                   CASE #tempRcvMsgTypeCase OF
                     #MQTT_MSG_TYPE_CONNACK:  // Statement section case 1
                       REGION RECEIVED_CONACK_PACKET    
                         #tempTrcvBufferPos += 1;
                         IF #statRcvBuffer[#tempTrcvBufferPos] = #REMAINING_LEN_2 //remainng Length must be 2;
                         THEN //
                           #tempTrcvBufferPos += 1;
                           //byte one is 0000 000X where X is if Session was set // so depending on clean session or not  evaluate answer of server
                           IF #statRcvBuffer[#tempTrcvBufferPos] = #MQTT_NO_SESSION_PRESENT THEN
                             #tempTrcvBufferPos += 1;
                             //VALID Answer, check code
                             IF #statRcvBuffer[#tempTrcvBufferPos] = #MQTT_CONNACK_ACCEPTED
                             THEN
                               //All good
                               #tempTrcvBufferPos += 1;
                               #tempMqttConnAckRcvStatus := #RESPONSE_GOOD; //evaluate in MQTT StateMachine Below the response
                             ELSE
                               //NOT VALID CONNACK from server shows session has a bad return code
                               #statStatus := #ERR_MQTT_CONNACK_RETURN_CODE_INVALID; // Set correct status that identifies error clearly
                               #statSubfunctionStatus := #statRcvBuffer[#tempTrcvBufferPos]; // Status or return value of called FBs, FCs and system blocks
                               #statFBErrorState := #statFBState; // Set error state number for diagnostic 
                               #statErrorUserCleared := TRUE;
                               // Exit loop
                               EXIT;
                             END_IF;
                           ELSE
                             //NOT VALID, CONNACK from server shows session present
                             #statStatus := #ERR_MQTT_CONNACK_INVALID_SESSION_FLAG; // Set correct status that identifies error clearly
                             #statSubfunctionStatus := #ERR_MQTT_CONNACK_INVALID_SESSION_FLAG; // Status or return value of called FBs, FCs and system blocks
                             #statFBErrorState := #statFBState; // Set error state number for diagnostic 
                             #statErrorUserCleared := TRUE;
                             // Exit loop
                             EXIT;
                           END_IF;
                         ELSE // We got a CONNACK paket, but remaining length was not 2 (Error)
                           #statStatus := #ERR_MQTT_REM_LEN_INVALID; // Set correct status that identifies error clearly
                           #statSubfunctionStatus := #ERR_MQTT_REM_LEN_INVALID; // Status or return value of called FBs, FCs and system blocks
                           #statFBErrorState := #statFBState; // Set error state number for diagnostic 
                           #statErrorUserCleared := TRUE;
                           // Exit loop
                           EXIT;
                         END_IF;
                       END_REGION RECEIVED_CONACK_PACKET  
                     #MQTT_MSG_TYPE_PINGRESP:
                       REGION RECEIVED_PINGRESP_PAKET
                         #tempTrcvBufferPos += 1;
                         IF #statRcvBuffer[#tempTrcvBufferPos] = #REMAINIG_LEN_0 //remainng Length must be 0;
                         THEN
                           #tempTrcvBufferPos += 1;
                           #tempMqttPingRspRcv := #RESPONSE_GOOD; //evaluate in MQTT StateMachine Below the response
                         ELSE// We got a Pingrsp paket, but remaining length was not 0 (Error)
                           #statStatus := #ERR_MQTT_REM_LEN_INVALID; // Set correct status that identifies error clearly
                           #statSubfunctionStatus := #ERR_MQTT_REM_LEN_INVALID; // Status or return value of called FBs, FCs and system blocks
                           #statFBErrorState := #statFBState; // Set error state number for diagnostic 
                           #statErrorUserCleared := TRUE;
                           // Exit loop
                           EXIT;
                         END_IF;
                       END_REGION RECEIVED_PINGRESP_PAKET
                     #MQTT_MSG_TYPE_PUBACK:
                       REGION RECEIVED_PUBACK_PAKET
                         #tempTrcvBufferPos += 1;
                         IF #statRcvBuffer[#tempTrcvBufferPos] = #REMAINING_LEN_2 //remainng Length must be 2;
                         THEN //
                           #tempTrcvBufferPos += 1;
                           #tempWordForSliceAddress := UINT_TO_WORD(#statPaketId);
                           IF #statRcvBuffer[#tempTrcvBufferPos] = #tempWordForSliceAddress.%B1 THEN
                             #tempTrcvBufferPos += 1;
                             IF #statRcvBuffer[#tempTrcvBufferPos] = #tempWordForSliceAddress.%B0 THEN
                               #tempTrcvBufferPos += 1;
                               #tempMqttPubAckRcv := #RESPONSE_GOOD;
                             ELSE
                               #tempTrcvBufferPos += 1;
                               #tempMqttPubAckRcv := #RESPONSE_PAKET_ID_INVALID;
                             END_IF;
                           ELSE
                             #tempTrcvBufferPos += 1;
                             #tempMqttPubAckRcv := #RESPONSE_PAKET_ID_INVALID;
                           END_IF;
                         ELSE
                           #statStatus := #ERR_MQTT_REM_LEN_INVALID; // Set correct status that identifies error clearly
                           #statSubfunctionStatus := #ERR_MQTT_REM_LEN_INVALID; // Status or return value of called FBs, FCs and system blocks
                           #statFBErrorState := #statFBState; // Set error state number for diagnostic 
                           #statErrorUserCleared := TRUE;
                           // Exit loop
                           EXIT;
                         END_IF;
                       END_REGION RECEIVED_PUBACK_PAKET
                     #MQTT_MSG_TYPE_PUBREC:
                       REGION RECEIVED_PUBREC_PAKET
                         #tempTrcvBufferPos += 1;
                         IF #statRcvBuffer[#tempTrcvBufferPos] = #REMAINING_LEN_2 //remainng Length must be 2;
                         THEN //
                           #tempTrcvBufferPos += 1;
                           #tempWordForSliceAddress := UINT_TO_WORD(#statPaketId);
                           IF #statRcvBuffer[#tempTrcvBufferPos] = #tempWordForSliceAddress.%B1 THEN
                             #tempTrcvBufferPos += 1;
                             IF #statRcvBuffer[#tempTrcvBufferPos] = #tempWordForSliceAddress.%B0 THEN
                               #tempTrcvBufferPos += 1;
                               #tempMqttPubRecRcv := #RESPONSE_GOOD;
                             ELSE
                               #tempTrcvBufferPos += 1;
                               #tempMqttPubRecRcv := #RESPONSE_PAKET_ID_INVALID;
                             END_IF;
                           ELSE
                             #tempTrcvBufferPos += 1;
                             #tempMqttPubRecRcv := #RESPONSE_PAKET_ID_INVALID;
                           END_IF;
                         ELSE
                           #statStatus := #ERR_MQTT_REM_LEN_INVALID; // Set correct status that identifies error clearly
                           #statSubfunctionStatus := #ERR_MQTT_REM_LEN_INVALID; // Status or return value of called FBs, FCs and system blocks
                           #statFBErrorState := #statFBState; // Set error state number for diagnostic 
                           #statErrorUserCleared := TRUE;
                           // Exit loop
                           EXIT;
                         END_IF;
                       END_REGION RECEIVED_PUBREC_PAKET
                     #MQTT_MSG_TYPE_PUBCOMP:
                       REGION RECEIVED_PUBCOMP_PAKET
                         #tempTrcvBufferPos += 1;
                         IF #statRcvBuffer[#tempTrcvBufferPos] = #REMAINING_LEN_2 //remainng Length must be 2;
                         THEN //
                           #tempTrcvBufferPos += 1;
                           #tempWordForSliceAddress := UINT_TO_WORD(#statPaketId);
                           IF #statRcvBuffer[#tempTrcvBufferPos] = #tempWordForSliceAddress.%B1 THEN
                             #tempTrcvBufferPos += 1;
                             IF #statRcvBuffer[#tempTrcvBufferPos] = #tempWordForSliceAddress.%B0 THEN
                               #tempTrcvBufferPos += 1;
                               #tempMqttPubCompRcv := #RESPONSE_GOOD;
                             ELSE
                               #tempTrcvBufferPos += 1;
                               #tempMqttPubCompRcv := #RESPONSE_PAKET_ID_INVALID;
                             END_IF;
                           ELSE
                             #tempTrcvBufferPos += 1;
                             #tempMqttPubCompRcv := #RESPONSE_PAKET_ID_INVALID;
                           END_IF;
                         ELSE
                           #statStatus := #ERR_MQTT_REM_LEN_INVALID; // Set correct status that identifies error clearly
                           #statSubfunctionStatus := #ERR_MQTT_REM_LEN_INVALID; // Status or return value of called FBs, FCs and system blocks
                           #statFBErrorState := #statFBState; // Set error state number for diagnostic 
                           #statErrorUserCleared := TRUE;
                           // Exit loop
                           EXIT;
                         END_IF;
                       END_REGION RECEIVED_PUBCOMP_PAKET
                     #MQTT_MSG_TYPE_SUBACK:
                       REGION RECEIVED_SUBACK_PAKET
                         #tempTrcvBufferPos += 1;
                         IF #statRcvBuffer[#tempTrcvBufferPos] = #REMAINING_LEN_3 //remainng Length must be 3;
                         THEN //
                           #tempTrcvBufferPos += 1;
                           #tempWordForSliceAddress := UINT_TO_WORD(#statPaketId);
                           IF #statRcvBuffer[#tempTrcvBufferPos] = #tempWordForSliceAddress.%B1 THEN
                             #tempTrcvBufferPos += 1;
                             IF #statRcvBuffer[#tempTrcvBufferPos] = #tempWordForSliceAddress.%B0 THEN
                               #tempTrcvBufferPos += 1;
                               IF #statRcvBuffer[#tempTrcvBufferPos] = #SUBSCRIBE_FAILURE THEN
                                 #tempTrcvBufferPos += 1;
                                 #tempMqttSubAckRcv := #RESPONSE_SUBSCRIBE_FAILED;
                               ELSE
                                 #tempTrcvBufferPos += 1;
                                 #tempMqttSubAckRcv := #RESPONSE_GOOD;
                               END_IF;
                             ELSE
                               #tempTrcvBufferPos += 1;
                               #tempMqttSubAckRcv := #RESPONSE_PAKET_ID_INVALID;
                             END_IF;
                           ELSE
                             #tempTrcvBufferPos += 1;
                             #tempMqttSubAckRcv := #RESPONSE_PAKET_ID_INVALID;
                           END_IF;
                         ELSE
                           #statStatus := #ERR_MQTT_REM_LEN_INVALID; // Set correct status that identifies error clearly
                           #statSubfunctionStatus := #ERR_MQTT_REM_LEN_INVALID; // Status or return value of called FBs, FCs and system blocks
                           #statFBErrorState := #statFBState; // Set error state number for diagnostic 
                           #statErrorUserCleared := TRUE;
                           // Exit loop
                           EXIT;
                         END_IF;
                       END_REGION RECEIVED_SUBACK_PAKET
                     #MQTT_MSG_TYPE_UNSUBACK:
                       REGION RECEIVED_UNSUBACK_PAKET
                         #tempTrcvBufferPos += 1;
                         IF #statRcvBuffer[#tempTrcvBufferPos] = #REMAINING_LEN_2 //remainng Length must be 2;
                         THEN //
                           #tempTrcvBufferPos += 1;
                           #tempWordForSliceAddress := UINT_TO_WORD(#statPaketId);
                           IF #statRcvBuffer[#tempTrcvBufferPos] = #tempWordForSliceAddress.%B1 THEN
                             #tempTrcvBufferPos += 1;
                             IF #statRcvBuffer[#tempTrcvBufferPos] = #tempWordForSliceAddress.%B0 THEN
                               #tempTrcvBufferPos += 1;
                               #tempMqttUnSubAckRcv := #RESPONSE_GOOD;
                             ELSE
                               #tempTrcvBufferPos += 1;
                               #tempMqttUnSubAckRcv := #RESPONSE_PAKET_ID_INVALID;
                             END_IF;
                           ELSE
                             #tempTrcvBufferPos += 1;
                             #tempMqttUnSubAckRcv := #RESPONSE_PAKET_ID_INVALID;
                           END_IF;
                         ELSE
                           #statStatus := #ERR_MQTT_REM_LEN_INVALID; // Set correct status that identifies error clearly
                           #statSubfunctionStatus := #ERR_MQTT_REM_LEN_INVALID; // Status or return value of called FBs, FCs and system blocks
                           #statFBErrorState := #statFBState; // Set error state number for diagnostic 
                           #statErrorUserCleared := TRUE;
                           // Exit loop
                           EXIT;
                         END_IF;
                       END_REGION RECEIVED_UNSUBACK_PAKET
                     #MQTT_MSG_TYPE_RCV_PUB_MESSAGE:
                       REGION RECEIVED_PUBLISH_PAKET_FROM_BROKER
                         //Received a message, start process.
                         //init
                         #tempMultiplierToDecode := #INIT_UDINT_1;
                         #statRcvMsgInternalStatus := #MSG_DECODE_STATUS_NO_NEW_MSG;
                         #statRcvMsgTotalLen := 0;
                         #statRcvMsgTopicLen := 0;
                         #statRcvMsgPayloadLen := 0;
                         //Check and store QoS for later use
                         IF (#statRcvBuffer[#tempTrcvBufferPos] AND #BIT_MASK_QOS) = #MQTT_MSG_TYPE_RCV_PUB_MESSAGE_QoS0
                         THEN
                           #statRcvMsgQoS := #MQTT_QOS_0;
                         ELSIF (#statRcvBuffer[#tempTrcvBufferPos] AND #BIT_MASK_QOS) = #MQTT_MSG_TYPE_RCV_PUB_MESSAGE_QoS1
                         THEN
                           #statRcvMsgQoS := #MQTT_QOS_1;
                         ELSIF (#statRcvBuffer[#tempTrcvBufferPos] AND #BIT_MASK_QOS) = #MQTT_MSG_TYPE_RCV_PUB_MESSAGE_QoS2
                         THEN
                           #statRcvMsgQoS := #MQTT_QOS_2;
                         ELSIF (#statRcvBuffer[#tempTrcvBufferPos] AND #BIT_MASK_QOS) = #MQTT_MSG_TYPE_RCV_PUB_MESSAGE_BAD
                         THEN
                           #statStatus := #ERR_MQTT_MALFORMED_QOS_RECEIVED; // Set correct status that identifies error clearly
                           #statSubfunctionStatus := #ERR_MQTT_MALFORMED_QOS_RECEIVED; // Status or return value of called FBs, FCs and system blocks
                           #statFBErrorState := #statFBState; // Set error state number for diagnostic 
                           #statErrorUserCleared := TRUE;
                           // Exit loop
                           EXIT;
                         END_IF;

                         //Calculate total publish len (topic,paketid,payload)
                         REPEAT
                           #tempTrcvBufferPos += 1; //Increment
                           #statRcvMsgTotalLen += BYTE_TO_UDINT((#statRcvBuffer[#tempTrcvBufferPos] AND #DEFAULT_MULTIPLIER_BYTE_127)) * #tempMultiplierToDecode;
                           #tempMultiplierToDecode *= #SEND_LEN_MULTIPLIER_UDINT_128;
                           IF (#tempMultiplierToDecode > #MAX_ALLOWED_PAKET_SIZE)
                           THEN//Throw error here // Malformed remain length.
                             #statStatus := #ERR_MQTT_REM_LEN_INVALID; // Set correct status that identifies error clearly
                             #statSubfunctionStatus := #ERR_MQTT_REM_LEN_INVALID; // Status or return value of called FBs, FCs and system blocks
                             #statFBErrorState := #statFBState; // Set error state number for diagnostic 
                             #statErrorUserCleared := TRUE;
                             // Exit loop
                             EXIT;
                           END_IF;
                         UNTIL ((#statRcvBuffer[#tempTrcvBufferPos] AND UDINT_TO_BYTE(#SEND_LEN_MULTIPLIER_UDINT_128)) = 0)
                         END_REPEAT;
                         #tempTrcvBufferPos += 1; //Increment
                         //#statIncPaketRemLen contains total paket len
                         //Save Topic Len
                         #tempWordForSliceAddress.%B1 := #statRcvBuffer[#tempTrcvBufferPos]; //MSB
                         #tempTrcvBufferPos += 1; //Increment
                         #tempWordForSliceAddress.%B0 := #statRcvBuffer[#tempTrcvBufferPos]; //LSB
                         #tempTrcvBufferPos += 1; //Increment
                         #statRcvMsgTopicLen := WORD_TO_UINT(#tempWordForSliceAddress);
                         //Set Payload len
                         IF #statRcvMsgQoS = #MQTT_QOS_0 THEN
                           //Payload Len is total Len minus topic len minus topic len info 
                           #statRcvMsgPayloadLen := #statRcvMsgTotalLen - #statRcvMsgTopicLen - #TWO_BYTE_LEN_INFO;
                         ELSE
                           //PayloadLen is total Len minus topic len minus topic len info minus paket Id len
                           #statRcvMsgPayloadLen := #statRcvMsgTotalLen - #statRcvMsgTopicLen - #TWO_BYTE_LEN_INFO - #TWO_BYTE_LEN_INFO;
                         END_IF;

                         //Clear Output message:
                         #receivedTopic := #EMPTY_WSTRING;
                         //Start receiving with topic
                         #statRcvMsgDecodeState := #MSG_DECODE_STATE_TOPIC;
                         //Start Topic at first character
                         #statRcvMsgTopicPos := #FIRST_CHARACTER;
                         //Start RcvMsg at first array element
                         #statRcvMsgPayloadPos := LOWER_BOUND(ARR := #receivedMsgPayload, DIM := #ONE_DIMENSION);
                         //Set Output for received len according to array dimension
                         #tempReceivedMsgDataArrayTotalLen := ABS(UPPER_BOUND(ARR := #receivedMsgPayload, DIM := #ONE_DIMENSION) - LOWER_BOUND(ARR := #receivedMsgPayload, DIM := #ONE_DIMENSION)) + #ARRAY_LEN_OFFSET_PLUS_1;
                         IF #statRcvMsgPayloadLen < #tempReceivedMsgDataArrayTotalLen THEN
                           #statRcvMsgDataLen := #statRcvMsgPayloadLen;
                         ELSE
                           #statRcvMsgDataLen := DINT_TO_UDINT(#tempReceivedMsgDataArrayTotalLen);
                         END_IF;
                       END_REGION RECEIVED_PUBLISH_PAKET_FROM_BROKER
                     #MQTT_MSG_DECODING:
                       REGION RECEIVED_PAKET_DECODE
                         CASE #statRcvMsgDecodeState OF
                           #MSG_DECODE_STATE_NO_PROCESSING: // NO Processing
                             ;
                           #MSG_DECODE_STATE_TOPIC:  // Statement section case 1
                             #tempReceivedTopicStringMaxLen := MAX_LEN(#receivedTopic);
                             //Copy Topic To WString Inout
                             IF #statRcvMsgTopicPos <= #tempReceivedTopicStringMaxLen THEN
                               #receivedTopic[#statRcvMsgTopicPos] := BYTE_TO_WCHAR(#statRcvBuffer[#tempTrcvBufferPos]);
                               #statRcvMsgTopicPos += 1;
                             ELSE
                               //Max String len reached.
                               #statRcvMsgInternalStatus := #MSG_DECODE_STATUS_TOPIC_TOO_LONG;
                             END_IF;
                             //decrement
                             #statRcvMsgTopicLen -= 1;
                             //increment
                             #tempTrcvBufferPos += 1;
                             //Check condition, if topic fully decoded:
                             IF #statRcvMsgTopicLen <= 0 THEN
                               //Decide what to do next:
                               IF #statRcvMsgQoS > #MQTT_QOS_0 THEN
                                 //NextStep Decode PaketID
                                 #statRcvMsgDecodeState := #MSG_DECODE_STATE_PAKET_ID_MSB;
                               ELSIF #statRcvMsgQoS = #MQTT_QOS_0 AND #statRcvMsgPayloadLen > 0 THEN
                                 //NextStep Decode Payload
                                 #statRcvMsgDecodeState := #MSG_DECODE_STATE_PAYLOAD;
                               ELSE
                                 // QoS=0 and no Payload => Done
                                 // Decoding complete
                                 #statRcvMsgDecodeState := #MSG_DECODE_STATE_NO_PROCESSING;
                                 //Set New message flag
                                 IF #statRcvMsgInternalStatus = #MSG_DECODE_STATUS_NO_NEW_MSG THEN
                                   //New message received ok
                                   #statRcvMsgStatus := #MSG_DECODE_STATUS_NEW_MSG_OK;
                                 ELSE
                                   //Message received, but Payload or Topic longer than inout data area
                                   #statRcvMsgStatus := #MSG_DECODE_STATUS_TOPIC_TOO_LONG;
                                 END_IF;
                               END_IF;
                             END_IF;
                           #MSG_DECODE_STATE_PAKET_ID_MSB:  // Decode PaketId MSB
                             //Copy PaketID
                             #statRcvMsgPaketId.%B1 := #statRcvBuffer[#tempTrcvBufferPos]; //MSB
                             #tempTrcvBufferPos += 1; //Increment
                             #statRcvMsgDecodeState := #MSG_DECODE_STATE_PAKET_ID_LSB;
                           #MSG_DECODE_STATE_PAKET_ID_LSB: // Decode PaketId LSB
                             //Copy PaketID
                             #statRcvMsgPaketId.%B0 := #statRcvBuffer[#tempTrcvBufferPos]; //LSB
                             #tempTrcvBufferPos += 1; //Increment
                             IF #statRcvMsgPayloadLen > 0 THEN
                               #statRcvMsgDecodeState := #MSG_DECODE_STATE_PAYLOAD;
                             ELSE
                               // Decoding complete
                               #statRcvMsgDecodeState := #MSG_DECODE_STATE_NO_PROCESSING;
                               //Set New message flag
                               IF #statRcvMsgInternalStatus = #MSG_DECODE_STATUS_NO_NEW_MSG THEN
                                 //New message received ok
                                 #statRcvMsgStatus := #MSG_DECODE_STATUS_NEW_MSG_OK;
                               ELSE
                                 //Message received, but Payload or Topic longer than inout data area
                                 #statRcvMsgStatus := #MSG_DECODE_STATUS_TOPIC_TOO_LONG;
                               END_IF;
                               // Send PubAck Msg
                               #statSendPubAckMsg := TRUE;
                             END_IF;
                           #MSG_DECODE_STATE_PAYLOAD:
                             #tempUpperBoundRcvMsgDataArray := UPPER_BOUND(ARR := #receivedMsgPayload, DIM := #ONE_DIMENSION);

                             IF #statRcvMsgPayloadPos <= #tempUpperBoundRcvMsgDataArray THEN
                               //Copy to output
                               #receivedMsgPayload[#statRcvMsgPayloadPos] := (#statRcvBuffer[#tempTrcvBufferPos]);
                               //Increment the pos
                               #statRcvMsgPayloadPos += 1;
                             ELSE
                               //Max Payload len reached, skip
                               #statRcvMsgInternalStatus := #MSG_DECODE_STATUS_PAYLOAD_TOO_LONG;
                             END_IF;
                             //Decrement msg payload len
                             #statRcvMsgPayloadLen -= 1;
                             //Increment Buffer Pos
                             #tempTrcvBufferPos += 1;
                             //Check condition, if payload fully decoded:
                             IF #statRcvMsgPayloadLen <= 0 THEN
                               // Decoding complete
                               #statRcvMsgDecodeState := #MSG_DECODE_STATE_NO_PROCESSING;
                               //Set New message flag
                               IF #statRcvMsgInternalStatus = #MSG_DECODE_STATUS_NO_NEW_MSG THEN
                                 //New message received ok
                                 #statRcvMsgStatus := #MSG_DECODE_STATUS_NEW_MSG_OK;
                               ELSE
                                 //Message received, but Payload or Topic longer than inout data area
                                 #statRcvMsgStatus := #MSG_DECODE_STATUS_PAYLOAD_TOO_LONG;
                               END_IF;
                               //Decide if a PUB ACK needs to be send
                               IF #statRcvMsgQoS > #MQTT_QOS_0 THEN
                                 // Send PubAck Msg
                                 #statSendPubAckMsg := TRUE;
                               END_IF;
                             END_IF;
                           ELSE
                             //else case
                             #statStatus := #ERR_UNDEFINED_STATE;
                             #statErrorUserCleared := TRUE;
                             ;
                         END_CASE;
                       END_REGION RECEIVED_PAKET_DECODE
                     ELSE // No Header found, SKIP entry of buffer:
                       #tempTrcvBufferPos += 1;
                   END_CASE;
                 END_WHILE;
               END_REGION TRCV_NEW_DATA
             END_IF;

             //Send an Publish Acknowledge Msg, if necessary
             REGION SEND_PUB_ACK_MSG_ON_SUBSCRIPTIONS
               //Send Acknowledgements to Subscribed messages, if requested (QoS =1)
               IF #statSendPubAckMsg = TRUE AND // send pub ack Request
                 #statMqttCommandState = #MQTT_COMMAND_STATE_NO_PROCESSING AND // no send job processing
                 #tempTsendcBusy = FALSE AND // tsendC is ready
                 #tempTsendcDone = FALSE // tsendC did not finished in this cycle
               THEN
                 //Set Pos
                 #statSendBufferPos := 0;
                 //Write Msg Type
                 #statSendBuffer[#statSendBufferPos] := #MQTT_MSG_TYPE_PUBACK;
                 #statSendBufferPos += 1;
                 //Write Msg Len
                 #statSendBuffer[#statSendBufferPos] := #REMAINING_LEN_2;
                 #statSendBufferPos += 1;
                 //Write Paket Id - first MSB then LSB
                 #statSendBuffer[#statSendBufferPos] := #statRcvMsgPaketId.%B1;
                 #statSendBufferPos += 1;
                 #statSendBuffer[#statSendBufferPos] := #statRcvMsgPaketId.%B0;
                 #statSendBufferPos += 1;
                 //Set Send Len:
                 #statTsendcLen := #statSendBufferPos;
                 //Send msg
                 #statTsendcReq := TRUE;
                 //Reset ack:
                 #statSendPubAckMsg := FALSE;
               END_IF;
             END_REGION SEND_PUB_ACK_MSG_ON_SUBSCRIPTIONS

             REGION MQTT_STATE_MACHINE
               CASE #statMqttConnectState OF
                 #MQTT_CONNECT_STATE_NO_PROCESSING:  // Statement section case 1
                   ;
                 #MQTT_CONNECT_STATE_BUILD_PAKET:  //
                   REGION BUILD_CONNECT_PAKET
                     //Remaining Length is the length of the variable header (10 bytes) plus the length of the Payload. 
                     //Max Len of Mqtt pakets is per Standard 268,435,455 Bytes (ff,ff,ff,7f)
                     //Calculate Remain Len will be 10 bytes
                     //plus Len of ClientId   (max 3*16382 WChars= 49.146 Bytes)
                     //plus Len of User (max 3*16382 WChars= 49.146 Bytes)
                     //plus Len of PW (max 3*16382 WChars= 49.146 Bytes)
                     //plus Len of WillTopic (max 3*16382 WChars= 49.146 Bytes)
                     //plus Len of WillMessage (max 65535 Bytes - as only 2 Bytes Len info is possible)
                     // = Total 262 119 Bytes


                     // Must obey, if not currently sending PubAck Msg on a subscription
                     // Else, try in the next cycle
                     IF #tempTsendcBusy = FALSE AND // tsendC is ready
                       #tempTsendcDone = FALSE AND  // tsendC did not finish in this cycle
                       #statTsendcReq = FALSE THEN // no request from pub ack request

                       //Only need to encode header once
                       IF #statPaketHeaderEncodeDone = FALSE THEN
                         // INIT
                         #statSendBufferPos := 0;
                         #statClientIdPos := #FIRST_CHARACTER;
                         #statClientIdEncodeState := #FIRST_ENCODING;

                         #statWillTopicEncodeState := #FIRST_ENCODING;
                         #statWillTopicPos := #FIRST_CHARACTER;

                         #statWillMessageEncodeState := #FIRST_ENCODING;
                         #statWillMessagePos := 0; // The Posistion for the WILL Message Array

                         #statUserNameEncodeState := #FIRST_ENCODING;
                         #statUserNamePos := #FIRST_CHARACTER;

                         #statPasswordEncodeState := #FIRST_ENCODING;
                         #statPasswordPos := #FIRST_CHARACTER;

                         #statSendPaketTotalRemLen := #CONNECT_HEADER_10BYTE_LEN;
                         #statClientIdLenUtf8Encoded := 0;
                         #statWillTopicLenUtf8Encoded := 0;
                         #statUsernameLenUtf8Encoded := 0;
                         #statPasswordLenUtf8Encoded := 0;
                         //End Init

                         // Encode Client ID Len
                         // Client ID must always be present
                         FOR #tempLoopCounter := #FIRST_CHARACTER TO LEN(#clientIdentifier) DO
                           "LMQTT_ConvertToUtf8"(character     := #clientIdentifier[#tempLoopCounter],
                                                 convertedUtf8 => #tempConvertedUtf8,
                                                 bytesUsed     => #tempBytesUsedUtf8,
                                                 error         => #tempErrorConvertUtf8,
                                                 status        => #tempStatusConvertUtf8);
                           #statClientIdLenUtf8Encoded := #statClientIdLenUtf8Encoded + #tempBytesUsedUtf8;
                         END_FOR;

                         #statSendPaketTotalRemLen := #statSendPaketTotalRemLen + #statClientIdLenUtf8Encoded + #TWO_BYTE_LEN_INFO;


                         IF #username <> #EMPTY_WSTRING
                         THEN
                           #tempUserFlag := TRUE;
                           FOR #tempLoopCounter := #FIRST_CHARACTER TO LEN(#username) DO
                             "LMQTT_ConvertToUtf8"(character     := #username[#tempLoopCounter],
                                                   convertedUtf8 => #tempConvertedUtf8,
                                                   bytesUsed     => #tempBytesUsedUtf8,
                                                   error         => #tempErrorConvertUtf8,
                                                   status        => #tempStatusConvertUtf8);
                             #statUsernameLenUtf8Encoded := #statUsernameLenUtf8Encoded + #tempBytesUsedUtf8;
                           END_FOR;
                           #statSendPaketTotalRemLen := #statSendPaketTotalRemLen + #statUsernameLenUtf8Encoded + #TWO_BYTE_LEN_INFO;
                         ELSE
                           #statUserNameEncodeState := #NOT_USED_NO_ENCODING;
                           #tempUserFlag := FALSE;
                         END_IF;

                         IF #password <> #EMPTY_WSTRING AND #username <> #EMPTY_WSTRING
                         THEN
                           #tempPasswordFlag := TRUE;
                           FOR #tempLoopCounter := #FIRST_CHARACTER TO LEN(#password) DO
                             "LMQTT_ConvertToUtf8"(character     := #password[#tempLoopCounter],
                                                   convertedUtf8 => #tempConvertedUtf8,
                                                   bytesUsed     => #tempBytesUsedUtf8,
                                                   error         => #tempErrorConvertUtf8,
                                                   status        => #tempStatusConvertUtf8);
                             #statPasswordLenUtf8Encoded := #statPasswordLenUtf8Encoded + #tempBytesUsedUtf8;
                           END_FOR;
                           #statSendPaketTotalRemLen := #statSendPaketTotalRemLen + #statPasswordLenUtf8Encoded + #TWO_BYTE_LEN_INFO;
                         ELSE
                           #statPasswordEncodeState := #NOT_USED_NO_ENCODING;
                           #tempPasswordFlag := FALSE;
                         END_IF;


                         IF #willtopic <> #EMPTY_WSTRING
                         THEN
                           #tempWillFlag := TRUE;
                           CASE #statWillQos OF
                             #MQTT_QOS_0:  // Statement section case 1
                               #tempWillQoS1 := FALSE;
                               #tempWillQoS2 := FALSE;
                             #MQTT_QOS_1:  // Statement section case 2 to 4
                               #tempWillQoS1 := TRUE;
                               #tempWillQoS2 := FALSE;
                             #MQTT_QOS_2:
                               #tempWillQoS1 := FALSE;
                               #tempWillQoS2 := True;
                             ELSE  // Statement section ELSE
                               ;
                           END_CASE;
                           FOR #tempLoopCounter := #FIRST_CHARACTER TO LEN(#willtopic) DO
                             // Statement section FOR
                             "LMQTT_ConvertToUtf8"(character     := #willtopic[#tempLoopCounter],
                                                   convertedUtf8 => #tempConvertedUtf8,
                                                   bytesUsed     => #tempBytesUsedUtf8,
                                                   error         => #tempErrorConvertUtf8,
                                                   status        => #tempStatusConvertUtf8);
                             #statWillTopicLenUtf8Encoded := #statWillTopicLenUtf8Encoded + #tempBytesUsedUtf8;
                           END_FOR;
                           //Add WillTopic Len and Will Message Len (and len info twice)
                           #statSendPaketTotalRemLen := #statSendPaketTotalRemLen + #statWillTopicLenUtf8Encoded + #statWillMessageCnt + (2 * #TWO_BYTE_LEN_INFO);
                         ELSE
                           #statWillTopicEncodeState := #NOT_USED_NO_ENCODING;
                           #statWillMessageEncodeState := #NOT_USED_NO_ENCODING;
                           #tempWillFlag := FALSE;
                           #statWillRetain := FALSE;
                           #tempWillQoS1 := FALSE;
                           #tempWillQoS2 := FALSE;
                         END_IF;

                         //Build Connect Telegram
                         //Fixed Header - Write Paket Type
                         #statSendBuffer[#statSendBufferPos] := #MQTT_MSG_TYPE_CONNECT; // 1 Byte
                         #statSendBufferPos += 1; // increment

                         //Write Remaining Paket Len info 
                         WHILE (#statSendPaketTotalRemLen > #DEFAULT_VALUE_ZERO)
                         DO//See MQTT Spec for explanation of this calculation
                           #statEncodedRemPaketLenAsByte := UDINT_TO_BYTE(#statSendPaketTotalRemLen MOD #SEND_LEN_MULTIPLIER_UDINT_128);
                           #statSendPaketTotalRemLen := #statSendPaketTotalRemLen / #SEND_LEN_MULTIPLIER_UDINT_128;
                           // if there are more data to encode, set the top bit of this byte
                           IF #statSendPaketTotalRemLen > #DEFAULT_VALUE_ZERO
                           THEN
                             // Do this and continue while loop
                             #statEncodedRemPaketLenAsByte := #statEncodedRemPaketLenAsByte OR UDINT_TO_BYTE(#SEND_LEN_MULTIPLIER_UDINT_128);
                             #statSendBuffer[#statSendBufferPos] := #statEncodedRemPaketLenAsByte;
                             #statSendBufferPos += 1;
                           ELSE
                             //do this and leave while loop
                             #statSendBuffer[#statSendBufferPos] := #statEncodedRemPaketLenAsByte;
                             #statSendBufferPos += 1;
                           END_IF;
                         END_WHILE;

                         //Build Connect Telegram
                         // Write Protocol name
                         #statSendBuffer[#statSendBufferPos] := #CONN_PROTOCOL_NAME_0;
                         #statSendBufferPos += 1;
                         #statSendBuffer[#statSendBufferPos] := #CONN_PROTOCOL_NAME_4;
                         #statSendBufferPos += 1;
                         #statSendBuffer[#statSendBufferPos] := CHAR_TO_BYTE('M');
                         #statSendBufferPos += 1;
                         #statSendBuffer[#statSendBufferPos] := CHAR_TO_BYTE('Q');
                         #statSendBufferPos += 1;
                         #statSendBuffer[#statSendBufferPos] := CHAR_TO_BYTE('T');
                         #statSendBufferPos += 1;
                         #statSendBuffer[#statSendBufferPos] := CHAR_TO_BYTE('T');
                         #statSendBufferPos += 1;
                         //Write Protocol Level
                         #statSendBuffer[#statSendBufferPos] := #CONN_PROTOCOL_MQTT_VERSION_3_1_1;
                         #statSendBufferPos += 1;
                         //Write Connect Flags
                         #statSendBuffer[#statSendBufferPos].%X0 := false;
                         #statSendBuffer[#statSendBufferPos].%X1 := True;
                         #statSendBuffer[#statSendBufferPos].%X2 := #tempWillFlag;
                         #statSendBuffer[#statSendBufferPos].%X3 := #tempWillQoS1;
                         #statSendBuffer[#statSendBufferPos].%X4 := #tempWillQoS2;
                         #statSendBuffer[#statSendBufferPos].%X5 := #statWillRetain;
                         #statSendBuffer[#statSendBufferPos].%X6 := #tempPasswordFlag;
                         #statSendBuffer[#statSendBufferPos].%X7 := #tempUserFlag;
                         #statSendBufferPos += 1;
                         //Write Keep Alive in sec
                         #tempWordForSliceAddress := UINT_TO_WORD(#connParam.keepAlive);
                         #statSendBuffer[#statSendBufferPos] := #tempWordForSliceAddress.%B1;
                         #statSendBufferPos += 1;
                         #statSendBuffer[#statSendBufferPos] := #tempWordForSliceAddress.%B0;
                         #statSendBufferPos += 1;

                         //Set To Complete this, can skip in further progess
                         #statPaketHeaderEncodeDone := TRUE;
                       END_IF;

                       // Payload
                       // These fields, if present, MUST appear in the order:
                       // Client Identifier, Will topic, Will message, User Name, password


                       //ClientIdentifier
                       IF #statSendBufferPos <= #MAX_BUFFER_LEN_SEND - #TWO_BYTE_LEN_INFO THEN
                         CASE #statClientIdEncodeState OF
                           #FIRST_ENCODING:  // Statement section case 1
                             //ADD len info into paket

                             #tempWordForSliceAddress := UINT_TO_WORD(#statClientIdLenUtf8Encoded);
                             #statSendBuffer[#statSendBufferPos] := #tempWordForSliceAddress.%B1; //MSB
                             #statSendBufferPos += 1;
                             #statSendBuffer[#statSendBufferPos] := #tempWordForSliceAddress.%B0; // LSB
                             #statSendBufferPos += 1;

                             FOR #tempLoopCounter := #statClientIdPos TO LEN(#clientIdentifier) DO
                               "LMQTT_ConvertToUtf8"(character     := #clientIdentifier[#tempLoopCounter],
                                                     convertedUtf8 => #tempConvertedUtf8,
                                                     bytesUsed     => #tempBytesUsedUtf8,
                                                     error         => #tempErrorConvertUtf8,
                                                     status        => #tempStatusConvertUtf8);

                               IF #statSendBufferPos + #tempBytesUsedUtf8 <= #MAX_BUFFER_LEN_SEND THEN
                                 #statClientIdPos += 1;
                                 CASE #tempBytesUsedUtf8 OF
                                   #UTF_1_BYTE_USED:  // Statement section case 1
                                     #statSendBuffer[#statSendBufferPos] := #tempConvertedUtf8.%B0;
                                     #statSendBufferPos += 1;
                                   #UTF_2_BYTE_USED:
                                     #statSendBuffer[#statSendBufferPos] := #tempConvertedUtf8.%B0;
                                     #statSendBufferPos += 1;
                                     #statSendBuffer[#statSendBufferPos] := #tempConvertedUtf8.%B1;
                                     #statSendBufferPos += 1;
                                   #UTF_3_BYTE_USED:  // Statement section case 2 to 4
                                     #statSendBuffer[#statSendBufferPos] := #tempConvertedUtf8.%B0;
                                     #statSendBufferPos += 1;
                                     #statSendBuffer[#statSendBufferPos] := #tempConvertedUtf8.%B1;
                                     #statSendBufferPos += 1;
                                     #statSendBuffer[#statSendBufferPos] := #tempConvertedUtf8.%B2;
                                     #statSendBufferPos += 1;
                                   ELSE  // Statement section ELSE
                                     ;
                                 END_CASE;
                               ELSE
                                 //When buffer full
                                 #statClientIdEncodeState := #SUBSEQUENT_ENCODING;
                                 EXIT;
                               END_IF;
                             END_FOR;
                             IF #statClientIdPos >= LEN(#clientIdentifier) THEN
                               #statClientIdEncodeState := #ENCODE_DONE;
                             END_IF;


                           #SUBSEQUENT_ENCODING:  // Statement section case 2 to 4
                             FOR #tempLoopCounter := #statClientIdPos TO LEN(#clientIdentifier) DO
                               "LMQTT_ConvertToUtf8"(character     := #clientIdentifier[#tempLoopCounter],
                                                     convertedUtf8 => #tempConvertedUtf8,
                                                     bytesUsed     => #tempBytesUsedUtf8,
                                                     error         => #tempErrorConvertUtf8,
                                                     status        => #tempStatusConvertUtf8);
                               IF #statSendBufferPos + #tempBytesUsedUtf8 <= #MAX_BUFFER_LEN_SEND THEN
                                 #statClientIdPos += 1;
                                 CASE #tempBytesUsedUtf8 OF
                                   #UTF_1_BYTE_USED:  // Statement section case 1
                                     #statSendBuffer[#statSendBufferPos] := #tempConvertedUtf8.%B0;
                                     #statSendBufferPos += 1;
                                   #UTF_2_BYTE_USED:
                                     #statSendBuffer[#statSendBufferPos] := #tempConvertedUtf8.%B0;
                                     #statSendBufferPos += 1;
                                     #statSendBuffer[#statSendBufferPos] := #tempConvertedUtf8.%B1;
                                     #statSendBufferPos += 1;
                                   #UTF_3_BYTE_USED:  // Statement section case 2 to 4
                                     #statSendBuffer[#statSendBufferPos] := #tempConvertedUtf8.%B0;
                                     #statSendBufferPos += 1;
                                     #statSendBuffer[#statSendBufferPos] := #tempConvertedUtf8.%B1;
                                     #statSendBufferPos += 1;
                                     #statSendBuffer[#statSendBufferPos] := #tempConvertedUtf8.%B2;
                                     #statSendBufferPos += 1;
                                   ELSE  // Statement section ELSE
                                     ;
                                 END_CASE;
                               ELSE
                                 //When buffer full
                                 EXIT;
                               END_IF;
                             END_FOR;
                             IF #statClientIdPos >= LEN(#clientIdentifier) THEN
                               #statClientIdEncodeState := #ENCODE_DONE;
                             END_IF;
                           ELSE  // Statement section ELSE
                             ; // IDLE / SKIP
                         END_CASE;
                       END_IF;

                       // Will Topic
                       // If the Will Flag is set to 1, the Will Topic is the next field in the payload. It must be > 0 Bytes

                       IF #statClientIdEncodeState = #ENCODE_DONE
                         AND #statSendBufferPos <= #MAX_BUFFER_LEN_SEND - #TWO_BYTE_LEN_INFO THEN
                         //When Client Id is encoded and buffer not full
                         //And willTopic is used
                         CASE #statWillTopicEncodeState OF
                           #FIRST_ENCODING:  // Statement section case 1
                             //ADD len info into paket

                             #tempWordForSliceAddress := UINT_TO_WORD(#statWillTopicLenUtf8Encoded);
                             #statSendBuffer[#statSendBufferPos] := #tempWordForSliceAddress.%B1; //MSB
                             #statSendBufferPos += 1;
                             #statSendBuffer[#statSendBufferPos] := #tempWordForSliceAddress.%B0; // LSB
                             #statSendBufferPos += 1;

                             FOR #tempLoopCounter := #statWillTopicPos TO LEN(#willtopic) DO
                               "LMQTT_ConvertToUtf8"(character     := #willtopic[#tempLoopCounter],
                                                     convertedUtf8 => #tempConvertedUtf8,
                                                     bytesUsed     => #tempBytesUsedUtf8,
                                                     error         => #tempErrorConvertUtf8,
                                                     status        => #tempStatusConvertUtf8);

                               IF #statSendBufferPos + #tempBytesUsedUtf8 <= #MAX_BUFFER_LEN_SEND THEN
                                 //Increment when successful
                                 #statWillTopicPos += 1;

                                 CASE #tempBytesUsedUtf8 OF
                                   #UTF_1_BYTE_USED:  // Statement section case 1
                                     #statSendBuffer[#statSendBufferPos] := #tempConvertedUtf8.%B0;
                                     #statSendBufferPos += 1;
                                   #UTF_2_BYTE_USED:
                                     #statSendBuffer[#statSendBufferPos] := #tempConvertedUtf8.%B0;
                                     #statSendBufferPos += 1;
                                     #statSendBuffer[#statSendBufferPos] := #tempConvertedUtf8.%B1;
                                     #statSendBufferPos += 1;
                                   #UTF_3_BYTE_USED:  // Statement section case 2 to 4
                                     #statSendBuffer[#statSendBufferPos] := #tempConvertedUtf8.%B0;
                                     #statSendBufferPos += 1;
                                     #statSendBuffer[#statSendBufferPos] := #tempConvertedUtf8.%B1;
                                     #statSendBufferPos += 1;
                                     #statSendBuffer[#statSendBufferPos] := #tempConvertedUtf8.%B2;
                                     #statSendBufferPos += 1;
                                   ELSE  // Statement section ELSE
                                     ;
                                 END_CASE;
                               ELSE
                                 //When buffer full
                                 #statWillTopicEncodeState := #SUBSEQUENT_ENCODING;
                                 EXIT;
                               END_IF;
                             END_FOR;

                             IF #statWillTopicPos >= LEN(#willtopic) THEN
                               #statWillTopicEncodeState := #ENCODE_DONE;
                             END_IF;

                           #SUBSEQUENT_ENCODING:  // Statement section case 2 to 4
                             FOR #tempLoopCounter := #statWillTopicPos TO LEN(#willtopic) DO
                               "LMQTT_ConvertToUtf8"(character     := #willtopic[#tempLoopCounter],
                                                     convertedUtf8 => #tempConvertedUtf8,
                                                     bytesUsed     => #tempBytesUsedUtf8,
                                                     error         => #tempErrorConvertUtf8,
                                                     status        => #tempStatusConvertUtf8);

                               IF #statSendBufferPos + #tempBytesUsedUtf8 <= #MAX_BUFFER_LEN_SEND THEN
                                 #statWillTopicPos += 1;
                                 CASE #tempBytesUsedUtf8 OF
                                   #UTF_1_BYTE_USED:  // Statement section case 1
                                     #statSendBuffer[#statSendBufferPos] := #tempConvertedUtf8.%B0;
                                     #statSendBufferPos += 1;
                                   #UTF_2_BYTE_USED:
                                     #statSendBuffer[#statSendBufferPos] := #tempConvertedUtf8.%B0;
                                     #statSendBufferPos += 1;
                                     #statSendBuffer[#statSendBufferPos] := #tempConvertedUtf8.%B1;
                                     #statSendBufferPos += 1;
                                   #UTF_3_BYTE_USED:  // Statement section case 2 to 4
                                     #statSendBuffer[#statSendBufferPos] := #tempConvertedUtf8.%B0;
                                     #statSendBufferPos += 1;
                                     #statSendBuffer[#statSendBufferPos] := #tempConvertedUtf8.%B1;
                                     #statSendBufferPos += 1;
                                     #statSendBuffer[#statSendBufferPos] := #tempConvertedUtf8.%B2;
                                     #statSendBufferPos += 1;
                                   ELSE  // Statement section ELSE
                                     ;
                                 END_CASE;
                               ELSE
                                 //When buffer full
                                 EXIT;
                               END_IF;
                             END_FOR;
                             IF #statWillTopicPos >= LEN(#willtopic) THEN
                               #statWillTopicEncodeState := #ENCODE_DONE;
                             END_IF;

                           ELSE  // Statement section ELSE
                             ;
                         END_CASE;
                       END_IF;

                       // Will Message
                       // This field consists OF a two Byte length followed BY the payload FOR the Will message expressed as a sequence bytes.

                       IF #statClientIdEncodeState = #ENCODE_DONE
                         AND #statWillTopicEncodeState = #ENCODE_DONE
                         AND #statSendBufferPos <= #MAX_BUFFER_LEN_SEND - #TWO_BYTE_LEN_INFO THEN
                         //When Client Id is encoded and buffer not full
                         CASE #statWillMessageEncodeState OF
                           #FIRST_ENCODING:  // Statement section case 1
                             //ADD len info into paket

                             #tempWordForSliceAddress := UINT_TO_WORD(#statWillMessageCnt);
                             #statSendBuffer[#statSendBufferPos] := #tempWordForSliceAddress.%B1; //MSB
                             #statSendBufferPos += 1;
                             #statSendBuffer[#statSendBufferPos] := #tempWordForSliceAddress.%B0; // LSB
                             #statSendBufferPos += 1;

                             #tempLowerWillMsgArrayBoundary := LOWER_BOUND(ARR := #willMsgPayload, DIM := #ONE_DIMENSION);

                             FOR #tempLoopCounter := #statWillMessagePos TO UINT_TO_DINT(#statWillMessageCnt - 1) DO
                               IF #statSendBufferPos <= #MAX_BUFFER_LEN_SEND THEN
                                 #statSendBuffer[#statSendBufferPos] := #willMsgPayload[#tempLowerWillMsgArrayBoundary + #tempLoopCounter];
                                 #statSendBufferPos += 1;
                                 //Increment when successful
                                 #statWillMessagePos += 1;
                               ELSE
                                 //When buffer full
                                 #statWillMessageEncodeState := #SUBSEQUENT_ENCODING;
                                 EXIT;
                               END_IF;
                             END_FOR;
                             // If everything was copied successfull
                             IF #statWillMessagePos >= #statWillMessageCnt THEN
                               #statWillMessageEncodeState := #ENCODE_DONE;
                             END_IF;

                           #SUBSEQUENT_ENCODING:  // Statement section case 2 to 4
                             #tempLowerWillMsgArrayBoundary := LOWER_BOUND(ARR := #willMsgPayload, DIM := #ONE_DIMENSION);

                             FOR #tempLoopCounter := #statWillMessagePos TO UINT_TO_DINT(#statWillMessageCnt - 1) DO
                               IF #statSendBufferPos <= #MAX_BUFFER_LEN_SEND THEN
                                 #statSendBuffer[#statSendBufferPos] := #willMsgPayload[#tempLowerWillMsgArrayBoundary + #tempLoopCounter];
                                 #statSendBufferPos += 1;
                                 //Increment when successful
                                 #statWillMessagePos += 1;
                               ELSE
                                 //When Buffer Full
                                 EXIT;
                               END_IF;
                             END_FOR;
                             // If everything was copied successfull
                             IF #statWillMessagePos >= #statWillMessageCnt THEN
                               #statWillMessageEncodeState := #ENCODE_DONE;
                             END_IF;


                           ELSE  // Statement section ELSE
                             ;
                         END_CASE;
                       END_IF;

                       // Username
                       // If the Username Flag is set to 1, the Username the next field in the payload. It must be > 0 Bytes

                       IF #statClientIdEncodeState = #ENCODE_DONE
                         AND (#statWillTopicEncodeState = #ENCODE_DONE OR #statWillTopicEncodeState = #NOT_USED_NO_ENCODING)
                         AND (#statWillMessageEncodeState = #ENCODE_DONE OR #statWillTopicEncodeState = #NOT_USED_NO_ENCODING)
                         AND #statSendBufferPos <= #MAX_BUFFER_LEN_SEND - #TWO_BYTE_LEN_INFO THEN
                         //When Will Topic and Will Message is encoded and buffer not full
                         CASE #statUserNameEncodeState OF
                           #FIRST_ENCODING:  // Statement section case 1
                             //ADD len info into paket

                             #tempWordForSliceAddress := UINT_TO_WORD(#statUsernameLenUtf8Encoded);
                             #statSendBuffer[#statSendBufferPos] := #tempWordForSliceAddress.%B1; //MSB
                             #statSendBufferPos += 1;
                             #statSendBuffer[#statSendBufferPos] := #tempWordForSliceAddress.%B0; // LSB
                             #statSendBufferPos += 1;

                             FOR #tempLoopCounter := #statUserNamePos TO LEN(#username) DO
                               "LMQTT_ConvertToUtf8"(character     := #username[#tempLoopCounter],
                                                     convertedUtf8 => #tempConvertedUtf8,
                                                     bytesUsed     => #tempBytesUsedUtf8,
                                                     error         => #tempErrorConvertUtf8,
                                                     status        => #tempStatusConvertUtf8);

                               IF #statSendBufferPos + #tempBytesUsedUtf8 <= #MAX_BUFFER_LEN_SEND THEN
                                 //Increment when successful
                                 #statUserNamePos += 1;

                                 CASE #tempBytesUsedUtf8 OF
                                   #UTF_1_BYTE_USED:  // Statement section case 1
                                     #statSendBuffer[#statSendBufferPos] := #tempConvertedUtf8.%B0;
                                     #statSendBufferPos += 1;
                                   #UTF_2_BYTE_USED:
                                     #statSendBuffer[#statSendBufferPos] := #tempConvertedUtf8.%B0;
                                     #statSendBufferPos += 1;
                                     #statSendBuffer[#statSendBufferPos] := #tempConvertedUtf8.%B1;
                                     #statSendBufferPos += 1;
                                   #UTF_3_BYTE_USED:  // Statement section case 2 to 4
                                     #statSendBuffer[#statSendBufferPos] := #tempConvertedUtf8.%B0;
                                     #statSendBufferPos += 1;
                                     #statSendBuffer[#statSendBufferPos] := #tempConvertedUtf8.%B1;
                                     #statSendBufferPos += 1;
                                     #statSendBuffer[#statSendBufferPos] := #tempConvertedUtf8.%B2;
                                     #statSendBufferPos += 1;
                                   ELSE  // Statement section ELSE
                                     ;
                                 END_CASE;
                               ELSE
                                 //When buffer full
                                 #statUserNameEncodeState := #SUBSEQUENT_ENCODING;
                                 EXIT;
                               END_IF;
                             END_FOR;

                             IF #statUserNamePos >= LEN(#username) THEN
                               #statUserNameEncodeState := #ENCODE_DONE;
                             END_IF;

                           #SUBSEQUENT_ENCODING:  // Statement section case 2 to 4
                             FOR #tempLoopCounter := #statUserNamePos TO LEN(#username) DO
                               "LMQTT_ConvertToUtf8"(character     := #username[#tempLoopCounter],
                                                     convertedUtf8 => #tempConvertedUtf8,
                                                     bytesUsed     => #tempBytesUsedUtf8,
                                                     error         => #tempErrorConvertUtf8,
                                                     status        => #tempStatusConvertUtf8);

                               IF #statSendBufferPos + #tempBytesUsedUtf8 <= #MAX_BUFFER_LEN_SEND THEN
                                 #statUserNamePos += 1;
                                 CASE #tempBytesUsedUtf8 OF
                                   #UTF_1_BYTE_USED:  // Statement section case 1
                                     #statSendBuffer[#statSendBufferPos] := #tempConvertedUtf8.%B0;
                                     #statSendBufferPos += 1;
                                   #UTF_2_BYTE_USED:
                                     #statSendBuffer[#statSendBufferPos] := #tempConvertedUtf8.%B0;
                                     #statSendBufferPos += 1;
                                     #statSendBuffer[#statSendBufferPos] := #tempConvertedUtf8.%B1;
                                     #statSendBufferPos += 1;
                                   #UTF_3_BYTE_USED:  // Statement section case 2 to 4
                                     #statSendBuffer[#statSendBufferPos] := #tempConvertedUtf8.%B0;
                                     #statSendBufferPos += 1;
                                     #statSendBuffer[#statSendBufferPos] := #tempConvertedUtf8.%B1;
                                     #statSendBufferPos += 1;
                                     #statSendBuffer[#statSendBufferPos] := #tempConvertedUtf8.%B2;
                                     #statSendBufferPos += 1;
                                   ELSE  // Statement section ELSE
                                     ;
                                 END_CASE;
                               ELSE
                                 //When buffer full
                                 EXIT;
                               END_IF;
                             END_FOR;
                             IF #statUserNamePos >= LEN(#username) THEN
                               #statUserNameEncodeState := #ENCODE_DONE;
                             END_IF;

                           ELSE  // Statement section ELSE
                             ;
                         END_CASE;
                       END_IF;

                       // Password
                       // If the Password Flag is set to 1, the Password the next field in the payload. It must be > 0 Bytes
                       //Password field contains 0 to 65535 bytes OF binary data prefixed with a two Byte length field which indicates the number OF bytes used

                       IF #statClientIdEncodeState = #ENCODE_DONE
                         AND (#statWillTopicEncodeState = #ENCODE_DONE OR #statWillTopicEncodeState = #NOT_USED_NO_ENCODING)
                         AND (#statWillMessageEncodeState = #ENCODE_DONE OR #statWillMessageEncodeState = #NOT_USED_NO_ENCODING)
                         AND (#statUserNameEncodeState = #ENCODE_DONE OR #statUserNameEncodeState = #NOT_USED_NO_ENCODING)
                         AND #statSendBufferPos <= #MAX_BUFFER_LEN_SEND - #TWO_BYTE_LEN_INFO THEN
                         //When Will Topic and Will Message is encoded and buffer not full
                         CASE #statPasswordEncodeState OF
                           #FIRST_ENCODING:  // Statement section case 1
                             //ADD len info into paket

                             #tempWordForSliceAddress := UINT_TO_WORD(#statPasswordLenUtf8Encoded);
                             #statSendBuffer[#statSendBufferPos] := #tempWordForSliceAddress.%B1; //MSB
                             #statSendBufferPos += 1;
                             #statSendBuffer[#statSendBufferPos] := #tempWordForSliceAddress.%B0; // LSB
                             #statSendBufferPos += 1;

                             FOR #tempLoopCounter := #statPasswordPos TO LEN(#password) DO
                               "LMQTT_ConvertToUtf8"(character     := #password[#tempLoopCounter],
                                                     convertedUtf8 => #tempConvertedUtf8,
                                                     bytesUsed     => #tempBytesUsedUtf8,
                                                     error         => #tempErrorConvertUtf8,
                                                     status        => #tempStatusConvertUtf8);

                               IF #statSendBufferPos + #tempBytesUsedUtf8 <= #MAX_BUFFER_LEN_SEND THEN
                                 //Increment when successful
                                 #statPasswordPos += 1;

                                 CASE #tempBytesUsedUtf8 OF
                                   #UTF_1_BYTE_USED:  // Statement section case 1
                                     #statSendBuffer[#statSendBufferPos] := #tempConvertedUtf8.%B0;
                                     #statSendBufferPos += 1;
                                   #UTF_2_BYTE_USED:
                                     #statSendBuffer[#statSendBufferPos] := #tempConvertedUtf8.%B0;
                                     #statSendBufferPos += 1;
                                     #statSendBuffer[#statSendBufferPos] := #tempConvertedUtf8.%B1;
                                     #statSendBufferPos += 1;
                                   #UTF_3_BYTE_USED:  // Statement section case 2 to 4
                                     #statSendBuffer[#statSendBufferPos] := #tempConvertedUtf8.%B0;
                                     #statSendBufferPos += 1;
                                     #statSendBuffer[#statSendBufferPos] := #tempConvertedUtf8.%B1;
                                     #statSendBufferPos += 1;
                                     #statSendBuffer[#statSendBufferPos] := #tempConvertedUtf8.%B2;
                                     #statSendBufferPos += 1;
                                   ELSE  // Statement section ELSE
                                     ;
                                 END_CASE;
                               ELSE
                                 //When buffer full
                                 #statPasswordEncodeState := #SUBSEQUENT_ENCODING;
                                 EXIT;
                               END_IF;
                             END_FOR;

                             IF #statPasswordPos >= LEN(#password) THEN
                               #statPasswordEncodeState := #ENCODE_DONE;
                             END_IF;

                           #SUBSEQUENT_ENCODING:  // Statement section case 2 to 4
                             FOR #tempLoopCounter := #statPasswordPos TO LEN(#password) DO
                               "LMQTT_ConvertToUtf8"(character     := #password[#tempLoopCounter],
                                                     convertedUtf8 => #tempConvertedUtf8,
                                                     bytesUsed     => #tempBytesUsedUtf8,
                                                     error         => #tempErrorConvertUtf8,
                                                     status        => #tempStatusConvertUtf8);

                               IF #statSendBufferPos + #tempBytesUsedUtf8 <= #MAX_BUFFER_LEN_SEND THEN
                                 #statPasswordPos += 1;
                                 CASE #tempBytesUsedUtf8 OF
                                   #UTF_1_BYTE_USED:  // Statement section case 1
                                     #statSendBuffer[#statSendBufferPos] := #tempConvertedUtf8.%B0;
                                     #statSendBufferPos += 1;
                                   #UTF_2_BYTE_USED:
                                     #statSendBuffer[#statSendBufferPos] := #tempConvertedUtf8.%B0;
                                     #statSendBufferPos += 1;
                                     #statSendBuffer[#statSendBufferPos] := #tempConvertedUtf8.%B1;
                                     #statSendBufferPos += 1;
                                   #UTF_3_BYTE_USED:  // Statement section case 2 to 4
                                     #statSendBuffer[#statSendBufferPos] := #tempConvertedUtf8.%B0;
                                     #statSendBufferPos += 1;
                                     #statSendBuffer[#statSendBufferPos] := #tempConvertedUtf8.%B1;
                                     #statSendBufferPos += 1;
                                     #statSendBuffer[#statSendBufferPos] := #tempConvertedUtf8.%B2;
                                     #statSendBufferPos += 1;
                                   ELSE  // Statement section ELSE
                                     ;
                                 END_CASE;
                               ELSE
                                 //When buffer full
                                 EXIT;
                               END_IF;
                             END_FOR;
                             IF #statPasswordPos >= LEN(#password) THEN
                               #statPasswordEncodeState := #ENCODE_DONE;
                             END_IF;

                           ELSE  // Statement section ELSE
                             ;
                         END_CASE;
                       END_IF;

                       //set Sendlen for TSendC Block

                       #statTsendcLen := #statSendBufferPos; // Buffer pos equals amount of elements in send array
                       //reset buffer pos
                       #statSendBufferPos := 0;
                       //enable Send Req
                       #statTsendcReq := TRUE;
                       //Set Watchdog
                       #statEnableTimerCommandWatchdog := TRUE;
                       //wait for send to be done
                       #statMqttConnectState := #MQTT_CONNECT_STATE_SEND_PAKET_WAIT_FOR_CONNACK;
                     END_IF;
                   END_REGION BUILD_CONNECT_PAKET
                 #MQTT_CONNECT_STATE_SEND_PAKET_WAIT_FOR_CONNACK:
                   REGION SEND_CONNECT_PAKET_WAIT_FOR_CONNACK
                     //check tsend status
                     IF NOT #tempTsendcBusy AND #tempTsendcStatus = #TSENDC_JOB_DONE THEN
                       IF (#statClientIdEncodeState = #ENCODE_DONE OR #statClientIdEncodeState = #NOT_USED_NO_ENCODING)
                         AND (#statWillTopicEncodeState = #ENCODE_DONE OR #statWillTopicEncodeState = #NOT_USED_NO_ENCODING)
                         AND (#statWillMessageEncodeState = #ENCODE_DONE OR #statWillMessageEncodeState = #NOT_USED_NO_ENCODING)
                         AND (#statUserNameEncodeState = #ENCODE_DONE OR #statUserNameEncodeState = #NOT_USED_NO_ENCODING)
                         AND (#statPasswordEncodeState = #ENCODE_DONE OR #statPasswordEncodeState = #NOT_USED_NO_ENCODING) THEN
                         //Encoding done all sent
                         #statPaketHeaderEncodeDone := FALSE;
                       ELSE
                         // More to Encode and send
                         #statEnableTimerCommandWatchdog := FALSE;
                         #statMqttConnectState := #MQTT_CONNECT_STATE_BUILD_PAKET;
                       END_IF;
                     END_IF;
                     //Check watchdog
                     IF #instTimerCommandWatchdog.Q THEN
                       #statEnableTimerCommandWatchdog := FALSE;
                       #statPaketHeaderEncodeDone := FALSE;
                       #statStatus := #ERR_MQTT_CONNECT_TIMEOUT; // Set correct status that identifies error clearly
                       #statSubfunctionStatus := #ERR_MQTT_CONNECT_TIMEOUT; // Status or return value of called FBs, FCs and system blocks
                       #statFBErrorState := #statFBState; // Set error state number for diagnostic 
                       #statErrorAutoCleared := TRUE;
                       #statMqttConnectState := #MQTT_CONNECT_STATE_BUILD_PAKET;
                     END_IF;

                     //Check Connect ACK paket
                     CASE #tempMqttConnAckRcvStatus OF
                       #NO_RESPONSE:  //  IDLE
                         ;
                       #RESPONSE_GOOD:  // Statement section case 2 to 4
                         //disable watchdog
                         #statEnableTimerCommandWatchdog := FALSE;
                         //Encoding done all sent
                         #statPaketHeaderEncodeDone := FALSE;
                         //Go to Connected
                         #statMqttConnectState := #MQTT_CONNECT_STATE_CONNECTED;
                         #statStatus := #STATUS_MQTT_CONNECTED;
                     END_CASE;
                   END_REGION REGION SEND_CONNECT_PAKET
                 #MQTT_CONNECT_STATE_CONNECTED:
                   REGION CONNECTED
                     //Check Rising edge of input commands
                     #tempCommandInput.%X0 := #tempPublish AND NOT #statPublishOld;
                     #tempCommandInput.%X1 := #tempSubscribe AND NOT #statSubscribeOld;
                     #tempCommandInput.%X2 := #tempUnsubscribe AND NOT #statUnsubscribeOld;

                     //Start the keepalive timer if used
                     #statEnableMqttKeepAliveTimer := #statMqttKeepAliveUsed;

                     //set status to connected after successfully executed job
                     IF #statStatus = #STATUS_JOB_EXECUTED THEN
                       #statStatus := #STATUS_MQTT_CONNECTED;
                     END_IF;

                     REGION MQTT_COMMANDS
                       //When state machine is ready for a new input then assign correct command
                       //Ping job can be overwritten by a command.
                         IF #tempCommandInput <> #NO_COMMAND
                         AND (#statMqttCommandState = #MQTT_COMMAND_STATE_NO_PROCESSING OR #statMqttCommandState = #MQTT_COMMAND_STATE_SEND_PING)
                       THEN
                         // New Input set, reset done flag
                         #statDone := FALSE;
                         #statMqttCommandState := BYTE_TO_DINT(#tempCommandInput);
                       END_IF;

                       CASE #statMqttCommandState OF
                         #MQTT_COMMAND_STATE_NO_PROCESSING:
                           //EMPTY STATE
                           ;
                         #MQTT_COMMAND_STATE_BUILD_PUBLISH:  // Statement section case 1
                           REGION PUBLISH_TO_TOPIC
                             //Remaining Length is the length of the variable header (TOPIC NAME + PacketID) plus the length of the Payload. 
                             //Max Len of Mqtt pakets is per Standard 268,435,455 Bytes (ff,ff,ff,7f)
                             //Calculate Remain Len will be
                             //Len of TOPIC   (max 3*16382 WChars= 49.146 Bytes)
                             //plus Len of PacketID (2 Bytes)
                             //plus Len of Payload (max 268,435,455 - 49.146 - 2 = 268.386.307 Bytes ca. 268 MB)
                             //Max Array / DB Len in TIA portal is around 16 MB or 16.777.216 Byte
                             //Set Status
                             #statStatus := #STATUS_MQTT_PUBLISH;

                             // Must obey, if not currently sending PubAck Msg on a subscription
                             // Else, try in the next cycle
                             IF #tempTsendcBusy = FALSE // when tsendC is ready
                               AND #tempTsendcDone = FALSE // tsendC did not finish in this cycle
                               AND #statTsendcReq = FALSE // TsendC request was not already requested by pub ack msg
                             THEN
                               IF #statPaketHeaderEncodeDone = FALSE THEN

                                 //Init
                                 #statSendPaketTotalRemLen := 0;
                                 #statSendBufferPos := 0;
                                 #statPublishQos := #qos;
                                 #statPublishMessageCnt := #publishMsgLen;
                                 #statPublishTopicEncodeState := #FIRST_ENCODING;
                                 #statPublishTopicPos := #FIRST_CHARACTER;
                                 #statPublishTopicLenUtf8Encoded := 0;
                                 #statPaketId += 1;//increment
                                 #statPaketIdEncoded := FALSE;
                                 #statPublishEncodeMessageState := #SUBSEQUENT_ENCODING; // No len info necessary so start directly at subsequent.
                                 #statPublishMessagePos := 0; // first array element

                                 //verify PayloadLen
                                 #tempMaxPublishDataArrayLen := ABS(UPPER_BOUND(ARR := #publishMsgPayload, DIM := #ONE_DIMENSION) - LOWER_BOUND(ARR := #publishMsgPayload, DIM := #ONE_DIMENSION)) + #ARRAY_LEN_OFFSET_PLUS_1;

                                 //check necessary boundaries
                                 IF #tempMaxPublishDataArrayLen < #statPublishMessageCnt THEN
                                   #statStatus := #ERR_CNT_EXCEEDS_ARRAY_DIMENSION; // Set correct status that identifies error clearly
                                   #statSubfunctionStatus := #ERR_CNT_EXCEEDS_ARRAY_DIMENSION; // Status or return value of called FBs, FCs and system blocks
                                   #statFBErrorState := #statFBState; // Set error state number for diagnostic 
                                   #statErrorAutoCleared := TRUE;
                                   #statMqttCommandState := #MQTT_COMMAND_STATE_NO_PROCESSING;
                                 ELSIF LEN(#mqttTopic) = #LEN_NULL THEN
                                   #statStatus := #ERR_MQTT_COMMAND_PUBLISH_TOPIC_INVALID; // Set correct status that identifies error clearly
                                   #statSubfunctionStatus := #ERR_MQTT_COMMAND_PUBLISH_TOPIC_INVALID; // Status or return value of called FBs, FCs and system blocks
                                   #statFBErrorState := #statFBState; // Set error state number for diagnostic 
                                   #statErrorAutoCleared := TRUE;
                                   #statMqttCommandState := #MQTT_COMMAND_STATE_NO_PROCESSING;
                                 ELSIF #statPublishQos > #MQTT_QOS_2 THEN
                                   #statStatus := #ERR_QOS_INVALID; // Set correct status that identifies error clearly
                                   #statSubfunctionStatus := #ERR_QOS_INVALID; // Status or return value of called FBs, FCs and system blocks
                                   #statFBErrorState := #statFBState; // Set error state number for diagnostic 
                                   #statErrorAutoCleared := TRUE;
                                   #statMqttCommandState := #MQTT_COMMAND_STATE_NO_PROCESSING;
                                 ELSE // All ok
                                   //Add amount of bytes for publish message
                                   #statSendPaketTotalRemLen := #statSendPaketTotalRemLen + #statPublishMessageCnt;
                                   //add publish  topic len
                                   FOR #tempLoopCounter := #FIRST_CHARACTER TO LEN(#mqttTopic) DO
                                     "LMQTT_ConvertToUtf8"(character     := #mqttTopic[#tempLoopCounter],
                                                           convertedUtf8 => #tempConvertedUtf8,
                                                           bytesUsed     => #tempBytesUsedUtf8,
                                                           error         => #tempErrorConvertUtf8,
                                                           status        => #tempStatusConvertUtf8);
                                     #statPublishTopicLenUtf8Encoded := #statPublishTopicLenUtf8Encoded + #tempBytesUsedUtf8;
                                   END_FOR;
                                   #statSendPaketTotalRemLen := #statSendPaketTotalRemLen + #statPublishTopicLenUtf8Encoded + #TWO_BYTE_LEN_INFO;

                                   //Build Publish Telegram
                                   //Fixed Header - Write Paket Type
                                   #statSendBuffer[#statSendBufferPos] := #MQTT_MSG_TYPE_PUBLISH;
                                   // Set DUP flag always to FALSE
                                   #statSendBuffer[#statSendBufferPos].%X3 := FALSE;
                                   // Set QoS Level
                                   CASE #statPublishQos OF
                                     #MQTT_QOS_0:  // Statement section case 0
                                       #statSendBuffer[#statSendBufferPos].%X2 := FALSE;
                                       #statSendBuffer[#statSendBufferPos].%X1 := FALSE;
                                     #MQTT_QOS_1:  // Statement section case 1
                                       #statSendBuffer[#statSendBufferPos].%X2 := FALSE;
                                       #statSendBuffer[#statSendBufferPos].%X1 := TRUE;
                                       //Add two byte len info for Mandatory packet ID
                                       #statSendPaketTotalRemLen := #statSendPaketTotalRemLen + #TWO_BYTE_LEN_INFO;
                                     #MQTT_QOS_2: // Statement section case 2
                                       #statSendBuffer[#statSendBufferPos].%X2 := TRUE;
                                       #statSendBuffer[#statSendBufferPos].%X1 := FALSE;
                                       //Add two byte len info for Mandatory packet ID
                                       #statSendPaketTotalRemLen := #statSendPaketTotalRemLen + #TWO_BYTE_LEN_INFO;
                                     ELSE
                                       ;
                                   END_CASE;
                                   //Set retain bit
                                   #statSendBuffer[#statSendBufferPos].%X0 := #retain;

                                   #statSendBufferPos += 1; // increment

                                   //Write Remaining Paket Len info 
                                   WHILE (#statSendPaketTotalRemLen > #DEFAULT_VALUE_ZERO)
                                   DO//See MQTT Spec for explanation of this calculation
                                     #statEncodedRemPaketLenAsByte := UDINT_TO_BYTE(#statSendPaketTotalRemLen MOD #SEND_LEN_MULTIPLIER_UDINT_128);
                                     #statSendPaketTotalRemLen := #statSendPaketTotalRemLen / #SEND_LEN_MULTIPLIER_UDINT_128;
                                     // if there are more data to encode, set the top bit of this byte
                                     IF #statSendPaketTotalRemLen > #DEFAULT_VALUE_ZERO
                                     THEN
                                       // Do this and continue while loop
                                       #statEncodedRemPaketLenAsByte := #statEncodedRemPaketLenAsByte OR UDINT_TO_BYTE(#SEND_LEN_MULTIPLIER_UDINT_128);
                                       #statSendBuffer[#statSendBufferPos] := #statEncodedRemPaketLenAsByte;
                                       #statSendBufferPos += 1;
                                     ELSE
                                       //do this and leave while loop
                                       #statSendBuffer[#statSendBufferPos] := #statEncodedRemPaketLenAsByte;
                                       #statSendBufferPos += 1;
                                     END_IF;
                                   END_WHILE;
                                   //When all done, set encode to true
                                   #statPaketHeaderEncodeDone := TRUE;
                                 END_IF;
                               END_IF;

                               //Header Encoded - now Topic, PacketId and Message need to be encoded.
                               IF #statPaketHeaderEncodeDone = TRUE THEN

                                 //Publish Topic
                                 IF #statSendBufferPos <= #MAX_BUFFER_LEN_SEND - #TWO_BYTE_LEN_INFO THEN
                                   CASE #statPublishTopicEncodeState OF
                                     #FIRST_ENCODING:  // Statement section case 1
                                       //ADD len info into paket

                                       #tempWordForSliceAddress := UINT_TO_WORD(#statPublishTopicLenUtf8Encoded);
                                       #statSendBuffer[#statSendBufferPos] := #tempWordForSliceAddress.%B1; //MSB
                                       #statSendBufferPos += 1;
                                       #statSendBuffer[#statSendBufferPos] := #tempWordForSliceAddress.%B0; // LSB
                                       #statSendBufferPos += 1;

                                       FOR #tempLoopCounter := #statPublishTopicPos TO LEN(#mqttTopic) DO
                                         "LMQTT_ConvertToUtf8"(character     := #mqttTopic[#tempLoopCounter],
                                                               convertedUtf8 => #tempConvertedUtf8,
                                                               bytesUsed     => #tempBytesUsedUtf8,
                                                               error         => #tempErrorConvertUtf8,
                                                               status        => #tempStatusConvertUtf8);

                                         IF #statSendBufferPos + #tempBytesUsedUtf8 <= #MAX_BUFFER_LEN_SEND THEN
                                           #statPublishTopicPos += 1;
                                           CASE #tempBytesUsedUtf8 OF
                                             #UTF_1_BYTE_USED:  // Statement section case 1
                                               #statSendBuffer[#statSendBufferPos] := #tempConvertedUtf8.%B0;
                                               #statSendBufferPos += 1;
                                             #UTF_2_BYTE_USED:
                                               #statSendBuffer[#statSendBufferPos] := #tempConvertedUtf8.%B0;
                                               #statSendBufferPos += 1;
                                               #statSendBuffer[#statSendBufferPos] := #tempConvertedUtf8.%B1;
                                               #statSendBufferPos += 1;
                                             #UTF_3_BYTE_USED:  // Statement section case 2 to 4
                                               #statSendBuffer[#statSendBufferPos] := #tempConvertedUtf8.%B0;
                                               #statSendBufferPos += 1;
                                               #statSendBuffer[#statSendBufferPos] := #tempConvertedUtf8.%B1;
                                               #statSendBufferPos += 1;
                                               #statSendBuffer[#statSendBufferPos] := #tempConvertedUtf8.%B2;
                                               #statSendBufferPos += 1;
                                             ELSE  // Statement section ELSE
                                               ;
                                           END_CASE;
                                         ELSE
                                           //When buffer full
                                           #statPublishTopicEncodeState := #SUBSEQUENT_ENCODING;
                                           EXIT;
                                         END_IF;
                                       END_FOR;
                                       IF #statPublishTopicPos >= LEN(#mqttTopic) THEN
                                         #statPublishTopicEncodeState := #ENCODE_DONE;
                                       END_IF;


                                     #SUBSEQUENT_ENCODING:  // Statement section case 2 to 4
                                       FOR #tempLoopCounter := #statPublishTopicPos TO LEN(#mqttTopic) DO

                                         "LMQTT_ConvertToUtf8"(character     := #mqttTopic[#tempLoopCounter],
                                                               convertedUtf8 => #tempConvertedUtf8,
                                                               bytesUsed     => #tempBytesUsedUtf8,
                                                               error         => #tempErrorConvertUtf8,
                                                               status        => #tempStatusConvertUtf8);
                                         IF #statSendBufferPos + #tempBytesUsedUtf8 <= #MAX_BUFFER_LEN_SEND THEN
                                           #statPublishTopicPos += 1;
                                           CASE #tempBytesUsedUtf8 OF
                                             #UTF_1_BYTE_USED:  // Statement section case 1
                                               #statSendBuffer[#statSendBufferPos] := #tempConvertedUtf8.%B0;
                                               #statSendBufferPos += 1;
                                             #UTF_2_BYTE_USED:
                                               #statSendBuffer[#statSendBufferPos] := #tempConvertedUtf8.%B0;
                                               #statSendBufferPos += 1;
                                               #statSendBuffer[#statSendBufferPos] := #tempConvertedUtf8.%B1;
                                               #statSendBufferPos += 1;
                                             #UTF_3_BYTE_USED:  // Statement section case 2 to 4
                                               #statSendBuffer[#statSendBufferPos] := #tempConvertedUtf8.%B0;
                                               #statSendBufferPos += 1;
                                               #statSendBuffer[#statSendBufferPos] := #tempConvertedUtf8.%B1;
                                               #statSendBufferPos += 1;
                                               #statSendBuffer[#statSendBufferPos] := #tempConvertedUtf8.%B2;
                                               #statSendBufferPos += 1;
                                             ELSE  // Statement section ELSE
                                               ;
                                           END_CASE;
                                         ELSE
                                           //When buffer full
                                           EXIT;
                                         END_IF;
                                       END_FOR;
                                       IF #statPublishTopicPos >= LEN(#mqttTopic) THEN
                                         #statPublishTopicEncodeState := #ENCODE_DONE;
                                       END_IF;
                                     ELSE  // SKIP if done
                                       ;
                                   END_CASE;
                                 END_IF;

                                 // Encode MessageID, when QOS > 0 and  Topic done and buffer not full
                                 IF #statPublishTopicEncodeState = #ENCODE_DONE
                                   AND #statPaketIdEncoded = FALSE
                                   AND #statSendBufferPos <= #MAX_BUFFER_LEN_SEND - #TWO_BYTE_LEN_INFO THEN
                                   // Check QoS - only necessary if QoS >0
                                   CASE #statPublishQos OF
                                     #MQTT_QOS_1:
                                       #tempWordForSliceAddress := UINT_TO_WORD(#statPaketId);
                                       #statSendBuffer[#statSendBufferPos] := #tempWordForSliceAddress.%B1; //MSB
                                       #statSendBufferPos += 1;
                                       #statSendBuffer[#statSendBufferPos] := #tempWordForSliceAddress.%B0; //LSB
                                       #statSendBufferPos += 1;
                                     #MQTT_QOS_2:
                                       #tempWordForSliceAddress := UINT_TO_WORD(#statPaketId);
                                       #statSendBuffer[#statSendBufferPos] := #tempWordForSliceAddress.%B1; //MSB
                                       #statSendBufferPos += 1;
                                       #statSendBuffer[#statSendBufferPos] := #tempWordForSliceAddress.%B0; //LSB
                                       #statSendBufferPos += 1;
                                     ELSE
                                       //No paket id to encode here
                                       ;
                                   END_CASE;
                                   //Finally:
                                   #statPaketIdEncoded := TRUE;
                                 END_IF;

                                 // Encode Payload, when  Topic done and PaketID Done and buffer not full
                                 IF #statPublishTopicEncodeState = #ENCODE_DONE
                                   AND #statPaketIdEncoded = TRUE
                                   AND #statSendBufferPos < #MAX_BUFFER_LEN_SEND THEN

                                   // Publish Message Encoding
                                   // This Contains the payload from the publish message expressed as a sequence bytes.
                                   CASE #statPublishEncodeMessageState OF
                                     #SUBSEQUENT_ENCODING:  // Statement section case 2 to 4
                                       #tempLowerBoundPublishDataArray := LOWER_BOUND(ARR := #publishMsgPayload, DIM := #ONE_DIMENSION);

                                       FOR #tempLoopCounter := #statPublishMessagePos TO UDINT_TO_DINT(#statPublishMessageCnt - 1) DO
                                         IF #statSendBufferPos <= #MAX_BUFFER_LEN_SEND THEN
                                           #statSendBuffer[#statSendBufferPos] := #publishMsgPayload[#tempLowerBoundPublishDataArray + #tempLoopCounter];
                                           #statSendBufferPos += 1;
                                           //Increment when successful
                                           #statPublishMessagePos += 1;
                                         ELSE
                                           //When Buffer Full
                                           EXIT;
                                         END_IF;
                                       END_FOR;
                                       // If everything was copied successfull
                                       IF #statPublishMessagePos >= #statPublishMessageCnt THEN
                                         #statPublishEncodeMessageState := #ENCODE_DONE;
                                       END_IF;
                                     ELSE  // Statement section ELSE
                                       ;
                                   END_CASE;
                                 END_IF;


                                 //set Sendlen for TSendC Block
                                 #statTsendcLen := #statSendBufferPos; // Buffer pos equals amount of elements in send array
                                 //reset buffer pos
                                 #statSendBufferPos := 0;
                                 //enable Send Req
                                 #statTsendcReq := TRUE;
                                 //Set Watchdog
                                 #statEnableTimerCommandWatchdog := TRUE;
                                 //wait for send to be done
                                 #statMqttCommandState := #MQTT_COMMAND_STATE_SEND_PUBLISH;
                               END_IF;
                             END_IF;

                           END_REGION PUBLISH_TO_TOPIC
                         #MQTT_COMMAND_STATE_SEND_PUBLISH:
                           REGION SEND_PUBLISH_WAIT_FOR_RESPONSE
                             //check tsend status
                             IF NOT #tempTsendcBusy AND #tempTsendcStatus = #TSENDC_JOB_DONE THEN
                               IF (#statPublishTopicEncodeState = #ENCODE_DONE)
                                 AND (#statPublishEncodeMessageState = #ENCODE_DONE) THEN
                                 //Encoding done all sent
                                 #statPaketHeaderEncodeDone := FALSE;
                                 //  with QoS = 0 Job done
                                 IF #statPublishQos = #MQTT_QOS_0 THEN
                                   // job done
                                   #statDone := TRUE;
                                   // go back to idle
                                   #statMqttCommandState := #MQTT_COMMAND_STATE_NO_PROCESSING;
                                   //reset Watchdog
                                   #statEnableTimerCommandWatchdog := FALSE;
                                   // Set Status back to connected
                                   #statStatus := #STATUS_JOB_EXECUTED;
                                 END_IF;
                               ELSE
                                 // More to Encode and send
                                 #statEnableTimerCommandWatchdog := FALSE;
                                 #statMqttCommandState := #MQTT_COMMAND_STATE_BUILD_PUBLISH;
                               END_IF;
                             END_IF;
                             //check watchdog
                             IF #instTimerCommandWatchdog.Q THEN
                               #statEnableTimerCommandWatchdog := FALSE;
                               #statStatus := #ERR_MQTT_COMMAND_SEND_TIMEOUT; // Set correct status that identifies error clearly
                               #statSubfunctionStatus := #ERR_MQTT_COMMAND_SEND_TIMEOUT; // Status or return value of called FBs, FCs and system blocks
                               #statFBErrorState := #statFBState; // Set error state number for diagnostic 
                               #statErrorAutoCleared := TRUE;
                               #statMqttCommandState := #MQTT_COMMAND_STATE_NO_PROCESSING;
                             END_IF;

